INTERFACE ITF_BaseControlElement_HMI_Connector_View EXTENDS ITF_BaseComponent_HMI_Connector_View

END_INTERFACE

(* stored: Version 1.1.0.1
   Itf ITF_BaseControlElement_HMI_Connector_View: Id {68ea5254-c6f9-0b12-28dd-4a241e11bb89} *)
